(* CoDeSys 2.3 export: Pack11string7SJ6xm0.EXP *)

(* POU SGL_Sismored/Sismored 4.0/Imported/Pack11string7SJ6xm0, ST *)
FUNCTION_BLOCK Pack11string7SJ6xm0
VAR_INPUT
	sInput1, sInput2, sInput3, sInput4, sInput5, sInput6, sInput7, sInput8, sInput9, sInput10, sInput11: STRING;
END_VAR
VAR_OUTPUT
	aOutput : ARRAY[1..11] OF STRING;
END_VAR
aOutput[1] := sInput1;
aOutput[2] := sInput2;
aOutput[3] := sInput3;
aOutput[4] := sInput4;
aOutput[5] := sInput5;
aOutput[6] := sInput6;
aOutput[7] := sInput7;
aOutput[8] := sInput8;
aOutput[9] := sInput9;
aOutput[10] := sInput10;
aOutput[11] := sInput11;

END_FUNCTION_BLOCK
